(* CODESYS project PLS-logikk.project

Project tree, tasks and I/O mapping:
  Device : CODESYS Control Win V3 x64, CODESYS, version 3.5.21.50
    application Application
      libraries: Standard, 3.5.22.0 (System); Util, 3.5.22.0 (System); VisuDialogs, * (System); VisuElemBase, * (System); OpenWeather Client SL, * (CODESYS)
      task MainTask (cyclic, interval t#20ms, priority 1) calls PLC_PRG
      task VISU_TASK (cyclic, interval 100 ms, priority 31) calls VisuElems.Visu_Prg
      global variables GVL
      program PLC_PRG [ST]
      Lists/
        text list ValgtPIDVerdier
        text list Bakkesensor
        text list Energiventil
        text list Pumpe
      function block FB_Belimo_Energy_Valve [ST]
      function block safety_maks [ST]
      visualisation System_Overview
      visualisation System_Web_Configuration
      function block pumpe_ventil [ST]
      function block prognose [ST]
    EnergiVentilKommunikasjon : Ethernet, CODESYS, version 4.2.0.0
        settings: IPAddress = [192,168,0,1]; SubnetMask = [255,255,255,0]; GatewayAddress = [0,0,0,0]; MACAddress = [16#00,16#00,16#00,16#00,16#00,16#00]; SaveCommunicationSettings = FALSE; IPAddress = [192,168,0,2]; SubnetMask = [255,255,255,0]; GatewayAddress = [0,0,0,0]
      ModbusTCP_Server_Device : ModbusTCP Server Device, CODESYS, version 4.5.0.0
          settings: UpdateableHolding = TRUE
          unmapped channels: Holding Registers, Input Registers
      Modbus_TCP_Client : Modbus TCP Client, CODESYS, version 4.5.0.0
        Modbus_TCP_Server : Modbus TCP Server, CODESYS, version 4.5.0.0
            settings: Unit-ID = 255; IPAddress = [127, 0, 0, 1]; Channel 0.Function Code = 3; Channel 0.Read Offset = 16#0000; Channel 0.Read Length = 100; Channel 0.Write Offset = 0; Channel 0.Write Length = 0; Channel 0.Cycle Time = 100; Channel 1.Function Code = 16; Channel 1.Read Offset = 0; Channel 1.Read Length = 0; Channel 1.Write Offset = 16#0000; Channel 1.Write Length = 100; Channel 1.Cycle Time = 100
            input  Application.PLC_PRG.EnergiVentilRegs : ARRAY[0..99] OF WORD  // Channel 0
            output Application.GVL.DefaultEnergiVentilRegs : ARRAY[0..99] OF WORD  // Channel 1
    PumpeKommunikasjon : Ethernet, CODESYS, version 4.2.0.0
        settings: IPAddress = [192,168,0,1]; SubnetMask = [255,255,255,0]; GatewayAddress = [0,0,0,0]; MACAddress = [16#00,16#00,16#00,16#00,16#00,16#00]; SaveCommunicationSettings = FALSE; IPAddress = [192,168,0,2]; SubnetMask = [255,255,255,0]; GatewayAddress = [0,0,0,0]
      ModbusTCP_Server_Device_1 : ModbusTCP Server Device, CODESYS, version 4.5.0.0
          settings: Port = 503; UpdateableHolding = TRUE
          unmapped channels: Holding Registers, Input Registers
      Modbus_TCP_Client_1 : Modbus TCP Client, CODESYS, version 4.5.0.0
        Modbus_TCP_Server_1 : Modbus TCP Server, CODESYS, version 4.5.0.0
            settings: Unit-ID = 255; IPAddress = [127, 0, 0, 1]; Port = 503; Channel 0.Function Code = 3; Channel 0.Read Offset = 16#0000; Channel 0.Read Length = 100; Channel 0.Write Offset = 0; Channel 0.Write Length = 0; Channel 0.Cycle Time = 100; Channel 1.Function Code = 16; Channel 1.Read Offset = 0; Channel 1.Read Length = 0; Channel 1.Write Offset = 16#0000; Channel 1.Write Length = 100; Channel 1.Cycle Time = 100
            input  Application.PLC_PRG.PumpeRegs : ARRAY[0..99] OF WORD  // Channel 0
            output Application.GVL.DefaultPumpeRegs : ARRAY[0..99] OF WORD  // Channel 1
  libraries: VisuSymbols, 4.5.0.0 (System)
  text list GlobalTextList
  AC_GENERATOR_DATA
*)

// Device/Application/GVL
{attribute 'qualified_only'}
VAR_GLOBAL RETAIN
	
//system
energiventil_type : INT := 0; // 0 = Belimo, 1 = Siemens
bakkesensor_type  : INT := 0; //
pumpe_type        : INT := 0; //


//Simulering/falske variabler
DefaultEnergiVentilRegs: ARRAY[0..99] OF WORD;
DefaultPumpeRegs: ARRAY[0..99] OF WORD;
END_VAR

// Device/Application/PLC_PRG
PROGRAM PLC_PRG
VAR RETAIN
	

	EnergiVentilRegs: ARRAY[0..99] OF WORD;
	PumpeRegs: ARRAY[0..99] OF WORD;
	
	//prognose 
	fbWeather		: OPW.ForecastWeather;
	fbWeatherBatch	: OPW.ForecastWeatherBatch;

    xExecute		: BOOL;
    xError			: opw.ERROR;
	xDone			: BOOL;
	xbusy			: BOOL;
	location		: OPW.GeoLocation := (
		ws_city		:= "Tomsø",
		ws_country_code	:= "no",
		s_latitude	:= '69.6489',
		s_longitude	:= '18.9551'
	);
	eUnits			: OPW.UNIT_OPTION := OPW.UNIT_OPTION.METRIC;
	sLangugeCode	: OPW.LANGUAGE_CODE := 'en';
	
    apiKey			: STRING := '622d42f5e83be24b2235ae08787d5a43';

    idx				: INT;
		
	tFetch			: TON;
	
	prognose_temp				: ARRAY[0..23] OF REAL;
	prognose_nedbor				: ARRAY[0..23] OF REAL;
	prognose_vind				: ARRAY[0..23] OF REAL;
	
	// FBs
	Belimovalve : FB_Belimo_Energy_Valve;
	ventil0_regulering: safety_maks;
	smelte_regulering: pumpe_ventil;
	prognose_regulering: prognose;
	
	//styres av bruker
	veksler_temp_grense			: REAL:= 5;
	temp_beskyttelse_omraade	: REAL:= 5;
	min_temp_grense				: REAL:= -5;
	hysterese_C					: REAL:=1.5;
	smelte_grense				: REAL:=1.5;
	frost_grense				: REAL:=3;
	energi_grense				: REAL:=40;
	fukt_grense					: REAL:=40;
	
	Kp_array : ARRAY [0..2] OF REAL := [5,5,5]; // 0 = ventil0, 1 = pmp, 2 = ventiler
	Ti_array : ARRAY [0..2] OF REAL := [10,100,100];
	Td_array : ARRAY [0..2] OF REAL := [0,0,0];
	
	antall_soner				: INT:=3;
	bestemt_pumpe				: REAL:=50;
	min_pumpe					: REAL:=0;
	max_pumpe					: REAL:=100;
	bestemt_aapning				: ARRAY[1..20] OF REAL:= [20(0)];
	bestemt0_aapning			: REAL:= 0;
	
	ventil_min					: ARRAY[1..20] OF REAL:= [20(0)];
	ventil_maks					: ARRAY[1..20] OF REAL:= [20(100)];
	
	ventil0_min					: REAL:= 0;
	ventil0_maks				: REAL:= 100;
	
	manuell						: BOOL := FALSE;
	manuell0					: BOOL:= FALSE;
	reset						: ARRAY[1..20] OF BOOL:= [20(FALSE)];
	reset0						: BOOL:= FALSE;
	min_temp_aktiv				: BOOL:= TRUE;
	predikt						: BOOL:= FALSE;
	forvarme_horisont           : REAL:= 6.0;
	
	//interne variabler
	i							: INT := 0;
	pumpe_sone					: INT;
	varme_tap					: REAL;
	flow_sone					: REAL;
	tur_sone					: REAL;
	//Simulering (tall er kun eksempler)
	C1							: REAL:= 50000.0; // J/K
	C2							: REAL:= 80000.0; // J/K
	rho							: REAL:= 1000.0;  // kg/m^3
	c_1							: REAL:= 4186.0;  // J/(kg*K)
	
	Tx							: REAL:= 80;	  // C
	
	G1							: REAL:= 2000.0;  // W/K
	G2							: REAL:= 500.0;   // W/K
	G3							: REAL:= 300.0;   // W/K
	
	x5							: REAL:= 55;
	
	v1 							: REAL:= -5.0;
    v2 							: REAL:= 10.0;
    v3 							: REAL:= 10.0;
    v4 							: REAL:= 10.0;
	
	dx1							: REAL;
	dx2							: REAL;
	dx3							: REAL;
	dx4							: REAL;
	dx5							: REAL;
	deltat						: REAL:= 0.1;	  // s

	//output
	standby						: ARRAY[1..20] OF BOOL:= [20(FALSE)];
	running						: ARRAY[1..20] OF BOOL:= [20(FALSE)];
	lockout						: ARRAY[1..20] OF BOOL:= [20(FALSE)];
	tilstand                    : ARRAY[1..20] OF STRING;
	ventil0_aapning_cmd			: REAL;
	ventil_aapning_cmd			: ARRAY[1..20] OF REAL;
	pumpe_hastighet_cmd			: REAL;


	//innput
	tur_temp					: REAL;
	retur_temp					: REAL;
	retur_temp2					: REAL;
	ute_temp					: REAL := -10;
	energi_forbruk				: REAL;
	bakke_temp 					: ARRAY[1..20] OF REAL:= [20(5)];
    bakke_fukt 					: ARRAY[1..20] OF REAL:= [20(0)];
	ventil0_aapning_rd			: REAL;
	ventil_aapning_rd			: ARRAY[1..20] OF REAL;
	pumpe_hastighet_rd			: REAL;	
	
END_VAR


//init
CASE GVL.energiventil_type OF
0: Belimovalve(HoldingRegs := EnergiVentilRegs);
tur_temp := Belimovalve.temp1_C;
retur_temp := Belimovalve.temp2_C;
END_CASE

fbWeather(
    xExecute := xExecute,
	sApiKey := apiKey,
	pGeoLocation := ADR(location),
	eUnits := eUnits,
	data := fbWeatherBatch);
	
xError:= fbWeather.eError;
xDone:= fbWeather.xDone;
xbusy:= fbWeather.xBusy;

IF fbWeather.xDone THEN

    FOR i := 0 TO 23 DO

        prognose_temp[i] := fbWeatherBatch.aHourlyData[i].r_temperature;
        prognose_nedbor[i] := fbWeatherBatch.aHourlyData[i].r_snow_last_hour;
        prognose_vind[i] := fbWeatherBatch.aHourlyData[i].r_wind_speed;

    END_FOR
	
	xExecute := FALSE;

END_IF

tFetch(IN := TRUE, PT := T#60M);

IF tFetch.Q THEN
    xExecute := TRUE;
    tFetch(IN := FALSE);
END_IF

prognose_regulering(
    prognose_temp       := prognose_temp,
    prognose_nedbor     := prognose_nedbor,
    prognose_vind       := prognose_vind,
    ute_temp_na         := ute_temp,
    bakke_temp          := bakke_temp,

    base_frost_grense   := frost_grense,
	base_fukt_grense	:= fukt_grense,
    base_smelte_grense  := smelte_grense,
    base_min_pumpe      := min_pumpe,
    base_max_pumpe      := max_pumpe,

    forvarme_horisont   := forvarme_horisont,		// Se 6 timer frem
    maks_onsket_temp_okning := 3.0,		// Hev setpunkt med x antall grader
    grense_endring         := 2.0,		// Senk grensen med x antall grader
    min_pumpe_okning     := 15.0,	// Øk pumpe hastigheten for at hver sone alltid får nok strøm
	aktiver_prediktiv	:= predikt);



ventil0_regulering(
	retur_temp:= retur_temp,
	temp_grense:= veksler_temp_grense,
	temp_beskyttelse_omraade:= temp_beskyttelse_omraade,
	forbruk:= energi_forbruk,
	forbruk_grense:= energi_grense,
	bestemt_ventil:= bestemt0_aapning,
	Kp:= Kp_array[0],
	Ti:= Ti_array[0],
	Td:= Td_array[0],
	min_ventil:= ventil0_min,
	max_ventil:= ventil0_maks,
	manuell:= manuell0,
	reset:= reset0);

	
ventil0_aapning_cmd:= ventil0_regulering.ventil;


FOR i := 1 TO antall_soner DO
    IF smelte_regulering.running[i] THEN
        pumpe_sone := i;
    END_IF
END_FOR
i:=0;

smelte_regulering(
	antall_soner:= antall_soner,
	bakke_temp:=bakke_temp,
	bakke_fukt:= bakke_fukt,
	frost_grense:= frost_grense,
	smelte_grense:= smelte_grense,
	fukt_grense:= fukt_grense,
	hysterese:= hysterese_C,
	min_temp_grense:= min_temp_grense,
	min_temp_aktiv:= min_temp_aktiv,
	Kp_pmp:= Kp_array[1],
	Tn_pmp:= Ti_array[1],
	Tv_pmp:= Td_array[1],
	Kp_vnt:= Kp_array[2],
	Tn_vnt:= Ti_array[2],
	Tv_vnt:= Td_array[2],
	manuell:= manuell,
	reset:= reset,
	bestemt_pumpe:= bestemt_pumpe,
	min_pumpe:= min_pumpe,
	max_pumpe:= max_pumpe,
	pumpe_sone:= pumpe_sone,
	bestemt_aapning:=bestemt_aapning,
	ventil_min:= ventil_min,
	ventil_maks:= ventil_maks);

standby:= smelte_regulering.standby;
running:= smelte_regulering.running;
lockout:= smelte_regulering.min_temp_lockout;
ventil_aapning_cmd:= smelte_regulering.ventil_cmd;
pumpe_hastighet_cmd:= smelte_regulering.pumpe_cmd;


FOR i := 1 TO antall_soner DO
	IF standby[i] THEN 
		tilstand[i] := 'i standby';
	ELSIF running[i] THEN 
		tilstand[i] := 'i running';
	ELSIF lockout[i] THEN 
		tilstand[i] := 'i lockout';
	ELSE
		tilstand[i] := 'av';
	END_IF
END_FOR

//simulering
	retur_temp:= ((1.0/ventil0_aapning_rd - 1.0) * tur_temp 
	+ ventil_aapning_rd[1] * v2 + ventil_aapning_rd[2] * ventil_aapning_rd[2] * v3 
	+ (1.0 - ventil_aapning_rd[1] - ventil_aapning_rd[1] * ventil_aapning_rd[2]) * v4);
	
	
dx1 := (1.0/C1) * ( pumpe_hastighet_rd * rho * c_1 * ( Tx - tur_temp) - G1 * (tur_temp - x5));

dx2 := (1.0/C2) * ( pumpe_hastighet_rd * ventil0_aapning_rd * ventil_aapning_rd[1] * rho * c_1 * (tur_temp - v2) + G2 * (v2 - bakke_temp[1]) - G3 * (bakke_temp[1] - ute_temp));

dx3 := (1.0/C2) * ( pumpe_hastighet_rd * ventil0_aapning_rd * ventil_aapning_rd[1] * ventil_aapning_rd[2] * rho * c_1 * (tur_temp - v3) + G2 * (v3 - bakke_temp[2]) - G3 * (bakke_temp[2] - ute_temp));

dx4 := (1.0/C2) * ( pumpe_hastighet_rd * ventil0_aapning_rd * (1.0 - ventil_aapning_rd[1] - ventil_aapning_rd[1]*ventil_aapning_rd[2]) * rho * c_1 * (tur_temp - v4) + G2 * (v4 - bakke_temp[3]) - G3 * (bakke_temp[3] - ute_temp));

dx5 := (1.0/C1) * ( pumpe_hastighet_rd * rho * c_1 * (retur_temp- x5) - G1 * (x5 - tur_temp));

//Numerisk integrasjon (Euler)
tur_temp := tur_temp + dx1 * deltat;
bakke_temp[1] := bakke_temp[1] + dx2 * deltat;
bakke_temp[2] := bakke_temp[2] + dx3 * deltat;
bakke_temp[3] := bakke_temp[3] + dx4 * deltat;
x5 := x5 + dx5 * deltat;

//Enkel beregning av temperaturen ut av hver sone
v2 := tur_temp - (tur_temp - bakke_temp[1]* pumpe_hastighet_rd * ventil0_aapning_rd * ventil_aapning_rd[1]);
v3 := tur_temp - (tur_temp - bakke_temp[1]* pumpe_hastighet_rd * ventil0_aapning_rd * ventil_aapning_rd[1] * ventil_aapning_rd[2]);
v4 := tur_temp - (tur_temp - bakke_temp[1]* pumpe_hastighet_rd * ventil0_aapning_rd * (1.0 - ventil_aapning_rd[1] - ventil_aapning_rd[1]*ventil_aapning_rd[2]));

END_PROGRAM

// Device/Application/prognose
FUNCTION_BLOCK prognose
VAR_INPUT
    // ── Værvarselsdata fra Python (oppdateres f.eks. hvert 30. minutt) ──────
    // Timevis prognose, indeks 0 = neste hele time, 23 = 24 timer frem
    prognose_temp       : ARRAY[0..23] OF REAL;		// Utetemperatur [°C]
    prognose_nedbor     : ARRAY[0..23] OF REAL;		// Nedbørsmengde [mm/t]
    prognose_vind       : ARRAY[0..23] OF REAL;		// Vindhastighet [m/s]

    // ── Nåtilstand ──────────────────────────────────────────────────────────
    ute_temp_na         : REAL;                     // Faktisk utetemperatur nå [°C]
    bakke_temp          : ARRAY[1..20] OF REAL;     // Faktisk bakketemperatur per sone [°C]

    // ── Brukerens grunninnstillinger (pass-through når prediktiv er av) ─────
    base_frost_grense   : REAL;     // Normal frostgrense for å gå i standby [°C]
    base_smelte_grense  : REAL;     // Normal smeltegrense for å gå i running [°C]
	base_fukt_grense	: REAL;		// Normal fuktgrense for å gå i running [%]
    base_min_pumpe      : REAL;     // Normalt minimum pumpesignal [%]
    base_max_pumpe      : REAL;     // Normalt maksimum pumpesignal [%]

    // ── Prediktive tuningsparametre ──────────────────────────────────────────
    forvarme_horisont   : REAL := 6.0;	// Hvor mange timer frem vi ser etter snøhendelser [t] Anbefalt: 3–8 t avhengig av termisk tregheten til banen
    maks_onsket_temp_okning : REAL := 3.0;	// Hvor mye vi hever onsket_temp under forvarmning [°C] Heves gradvis jo nærmere snøhendelsen er
    grense_endring         : REAL := 1.5;	// Hvor mye vi hever frost_grense / smelte_grense for tidlig aktivering [°C] Gjør at sonene starter standby/running litt tidligere enn normalt
    min_pumpe_okning     : REAL := 15.0;	// Ekstra minimum pumpeprosent under forvarmning [%] Hindrer at pumpen stopper helt mens banen forvarmes
    vind_kjoele_faktor  : REAL := 0.16;	// Justeringsfaktor for vindavkjøling (standard vindkjøleformel) Følger wind chill index
    aktiver_prediktiv   : BOOL := FALSE;	// Slå prediktiv styring av/på
END_VAR

VAR_OUTPUT
    // ── Justerte setpunkter – kobles direkte til smelte_regulering ──────────
    ut_frost_grense     : REAL;     // Justert frostgrense
    ut_smelte_grense    : REAL;     // Justert smeltegrense
	ut_fukt_grense		: REAL;		// Justert fuktgrense
    ut_min_pumpe        : REAL;     // Justert minimum pumpe
    ut_max_pumpe        : REAL;     // Uendret, sendt videre

    // ── Statusinformasjon ────────────────────────────────────────────────────
    snoe_risiko         : REAL;     // Beregnet snørisiko 0–100
    timer_til_sno		: REAL;     	// Timer til første forventede snøhendelse (-1 = ingen)
    forvarme_aktiv		: BOOL;     // TRUE mens prediktiv forvarmning pågår
    forvarme_intensitet : REAL;     // 0–100 % — hvor aggressivt vi forvarmer
    vind_prognose_temp	: ARRAY[0..23] OF REAL;     	// Beregnet vindkjølt temperatur [°C]
END_VAR

VAR
    i                   : INT;

    // Interne beregningsvariabler
    forste_sno_time    : REAL;     // Indeks (timer) til første snøhendelse
    sno_funnet         : BOOL;
    sum_sno_mm         : REAL;     // Total forventet snønedbør innen horisonten
    min_prognose_temp   : REAL;     // Laveste temperatur innen horisonten

    intensitet_raa      : REAL;     // Ubehandlet intensitetsverdi 0–1
    tid_igjen_normert   : REAL;     // 0 = snøen er her, 1 = akkurat innenfor horisont
    temp_bidrag         : REAL;
    nedbor_bidrag       : REAL;
    vind_bidrag         : REAL;
    horisont_heltall    : INT;      // Horisont avrundet til heltall timer (maks 23)
END_VAR

//Beskytte mot dårlig input
IF forvarme_horisont < 1.0 THEN forvarme_horisont := 1.0; END_IF
IF forvarme_horisont > 23.0 THEN forvarme_horisont := 23.0; END_IF
horisont_heltall := REAL_TO_INT(forvarme_horisont);

//Finner første snøhendelse, total snø, laveste temp
sno_funnet      := FALSE;
forste_sno_time := -1.0;
sum_sno_mm      := 0.0;
min_prognose_temp := prognose_temp[0];

FOR i := 0 TO horisont_heltall DO
	//Regner ut hvor mye vinden påvirker temperaturen
	IF prognose_vind[i] > 1.3 AND prognose_temp[i] < 10.0 THEN
    	vind_prognose_temp[i] := 13.12
					 			+ 0.6215  * prognose_temp[i]
								- 11.37   * EXPT(prognose_vind[i] * 3.6, vind_kjoele_faktor)
								+ 0.3965  * prognose_temp[i] * EXPT(prognose_vind[i] * 3.6, vind_kjoele_faktor);
	ELSE
		vind_prognose_temp[i] := prognose_temp[i];
	END_IF

    // Registrer laveste temperatur 
    IF vind_prognose_temp[i] < min_prognose_temp THEN
        min_prognose_temp := vind_prognose_temp[i];
    END_IF

    // Finner ut om det kommer snø basert på forventet nedbør og temperatur
    IF (vind_prognose_temp[i] <= 0 AND prognose_nedbor[i] > 0.1) THEN

        sum_sno_mm := sum_sno_mm + prognose_nedbor[i];

        IF NOT sno_funnet THEN
            forste_sno_time := INT_TO_REAL(i);
            sno_funnet := TRUE;
        END_IF
	END_IF
END_FOR

timer_til_sno := forste_sno_time;  // -1 hvis ingen hendelse funnet

// Risiko bergening  (0–100)%
//    Tre bidrag vektet sammen:
//      – Temperaturrisiko : lavere temp → høyere risiko
//      – Nedbørsrisiko    : mer nedbør → høyere risiko
//      – Vindrisiko       : sterk vind forsterker nedkjøling

// Temperaturbidrag: 0 ved +5 °C eller mer, 100 ved -10 °C eller mindre
temp_bidrag := LIMIT(0.0, (5.0 - min_prognose_temp) / 15.0 * 100.0, 100.0);

// Nedbørsbidrag: 0 ved 0 mm eller mindre, 100 ved ≥10 mm total nedbør i vinduet
nedbor_bidrag := LIMIT(0.0, sum_sno_mm / 10.0 * 100.0, 100.0);

// Vindbidrag: 0 ved 0 m/s eller mindre, 100 ved ≥15 m/s
vind_bidrag := LIMIT(0.0, prognose_vind[0] / 15.0 * 100.0, 100.0);

// Vektet sum  (temperatur teller mest for bakke-systemet)
snoe_risiko := LIMIT(0.0,
    0.50 * temp_bidrag
  + 0.35 * nedbor_bidrag
  + 0.15 * vind_bidrag,
  100.0);

// Beregner forvarme intensitet  (0–1 brukes videre, 0–100 for å vise bruker)
//    Intensiteten trappes opp jo nærmere snøhendelsen vi er.
//    Ingen snøhendelse innen horisonten gjør at intensitet = 0
intensitet_raa := 0.0;

IF aktiver_prediktiv AND sno_funnet THEN
    // Normaliser: 0 = snøen er her, 1 = akkurat på horisonten
    tid_igjen_normert := LIMIT(0.0, forste_sno_time / forvarme_horisont, 1.0);

    // Lineær opptrapping: tidligst = 30 % intensitet, nærmer seg = 100 %
    intensitet_raa := LIMIT(0.0, 1.0 - (0.7 * tid_igjen_normert), 1.0);

    // I tillegg skaleres med risikoscoren (sterk storm → enda mer aggressiv)
    intensitet_raa := intensitet_raa * (0.5 + 0.5 * (snoe_risiko / 100.0));
END_IF

forvarme_aktiv      := intensitet_raa > 0.0;
forvarme_intensitet := LIMIT(0.0, intensitet_raa * 100.0, 100.0);

// Justerer sett punkter
//    Alle utganger faller tilbake til brukerens basisverdier når prediktiv er av
//    eller ingen snø er forventet.
IF aktiver_prediktiv AND forvarme_aktiv THEN

    // Hev frost-, fukt- og smeltegrensene litt slik at sonene aktiverer seg tidligere
    ut_frost_grense  := base_frost_grense  + grense_endring * intensitet_raa;
    ut_smelte_grense := base_smelte_grense + grense_endring * intensitet_raa;
	ut_fukt_grense   := base_fukt_grense   - base_fukt_grense * intensitet_raa;

    // Hev minimum pumpe for å hindre pumpen i å stoppe under forvarmning
    ut_min_pumpe     := LIMIT(base_min_pumpe,
                              base_min_pumpe + min_pumpe_okning * forvarme_intensitet,
                              base_max_pumpe * 0.8);
    ut_max_pumpe     := base_max_pumpe;

ELSE
    // Pass-through når prediktiv styring gjør ingenting (enten ved avskrudd eller ved ingen forventet snø)
    ut_frost_grense  := base_frost_grense;
    ut_smelte_grense := base_smelte_grense;
	ut_fukt_grense	 := base_fukt_grense;
    ut_min_pumpe     := base_min_pumpe;
    ut_max_pumpe     := base_max_pumpe;
END_IF

END_FUNCTION_BLOCK

// Device/Application/FB_Belimo_Energy_Valve
FUNCTION_BLOCK FB_Belimo_Energy_Valve
VAR_INPUT
	HoldingRegs : ARRAY[0..99] OF WORD; // map til Modbus Holding Registers
END_VAR
VAR_OUTPUT
	RelPos_pct : REAL;
    Flow_lps : REAL;
    Temp1_C : REAL;
    Temp2_C : REAL;
    DeltaT_K : REAL;
    Energy_kWh : REAL;
END_VAR
VAR
	rawLow : WORD;
    rawHigh : WORD;
    raw32 : DWORD;
END_VAR


//Konvertering
RelPos_pct := TO_REAL(HoldingRegs[4]) * 0.01;

Flow_lps := TO_REAL(HoldingRegs[7]) * 0.001;

Temp1_C := TO_REAL(HoldingRegs[19]) * 0.01; //vi sier at dette er tur temp for enkelhet, kunne ha vært invertert

Temp2_C := TO_REAL(HoldingRegs[21]) * 0.01;// retur temp

DeltaT_K := TO_REAL(HoldingRegs[23]) * 0.01;// diff mellom tur og retur

END_FUNCTION_BLOCK

// Device/Application/safety_maks
FUNCTION_BLOCK safety_maks
VAR_INPUT
	retur_temp                  : REAL;  // Retur temperatur sensor rett før varmeveksler og etter treveis ventil
    temp_grense                 : REAL;  // Temperatur hvor man må begynne å ta hensyn til sikkerheten rundt varmevekslere
    temp_beskyttelse_omraade    : REAL;  // Området under tem_grense for helt stengt ventil
                                         // Ved temp_grense - temp_beskyttelse_omraade blir ventil = 100%

    forbruk                     : REAL;  // Nåverende energi forbruk (kW)
    forbruk_grense              : REAL;  // Maks tillat energi forbruk (kW)

    bestemt_ventil              : REAL;  // Hvor stor åpning ventilen har i manuell modus
    Kp                          : REAL;  
    Ti                          : REAL;
    Td                          : REAL;
    min_ventil                  : REAL; // Når ventilen går fullt til smelte soner
    max_ventil                  : REAL; // Når ventilen går fullt tilbake til varmeveklser
    manuell                     : BOOL;
    reset                       : BOOL;
END_VAR
VAR_OUTPUT
    ventil                      : REAL;	// Signal som bestemmer ventil possisjon
    beskyttelse_aktiv           : BOOL; // På når beskyttelse modus er aktiv
    beskyttelse_faktor          : REAL; // Faktor som sier hvor mye beskytelsen er på (0.0 beskyttelsen er av, 1.0 beskyttelsen sender alt tilbake til varmeveksler
END_VAR
VAR
	offset                      : REAL := 0;
    pid                         : PID;
    Max_tillatt                : REAL;  // Min valve position allowed by protection
END_VAR

// BESKYTT MOT DÅRLIG INNGANG
// Forhindrer divisjon med null hvis område ikke er konfigurert
IF temp_beskyttelse_omraade <= 0.0 THEN
    temp_beskyttelse_omraade := 1.0;
END_IF

//bestemmer hvor mye beskyttelse som skla være på
IF retur_temp >= temp_grense THEN
    beskyttelse_faktor := 0.0;
ELSIF retur_temp <= (temp_grense - temp_beskyttelse_omraade) THEN
    beskyttelse_faktor := 1.0;
ELSE
    beskyttelse_faktor := (temp_grense - retur_temp) / temp_beskyttelse_omraade;
END_IF;

//setter beskytelses indikator på hvis det er mer enn 0.0 beskytelse
beskyttelse_aktiv := beskyttelse_faktor > 0.0;

//definerer en minimums grense tillat slik at pid-regulatoren ikke kan sende mer til smelte soner enn trygt
Max_tillatt := max_ventil - (beskyttelse_faktor * (max_ventil - min_ventil));

//pid for å regulere energi forbruk
pid(
    ACTUAL      := forbruk,
    SET_POINT   := forbruk_grense,
    KP          := Kp,
    TN          := Ti,
    TV          := Td,
    Y_MANUAL    := bestemt_ventil,
    Y_OFFSET    := offset,
    Y_MIN       := min_ventil,
    Y_MAX       := max_tillatt,
    MANUAL      := manuell,
    RESET       := reset);

ventil := LIMIT(Min_ventil, pid.Y, max_tillatt);

//når ventil er 100% går all strøm til smelte sonene og når ventil er 0% vil alø strøm gå igjennom tre veis ventilen og tilbake til varmeveksleren

END_FUNCTION_BLOCK

// Device/Application/pumpe_ventil
FUNCTION_BLOCK pumpe_ventil
VAR_INPUT
	
	antall_soner        : INT;	//Hvor mange soner du ønsker å regulere
    bakke_temp          : ARRAY[1..20] OF REAL;	//Array av alle bakke temp målinger
    bakke_fukt          : ARRAY[1..20] OF REAL;	//Array av alle bakke fukt målinger
	
    frost_grense        : REAL;	//Nedre grense for å starte tining
    smelte_grense       : REAL;	//Øvre grense for å starte tining
    fukt_grense         : REAL;	//Grense for hvor mye fukt for å starte tining
    hysterese           : REAL;	//Ekstra ledd for å forhindre hopping mellom tilstander
	
	min_temp_grense     : REAL;	//Under denne tempen vil systemet gå i lockout
    min_temp_aktiv      : BOOL; //Velg om du vil inkludere lockout
	
	Kp_pmp              : REAL;	//Kp-verdi for pumpe
    Tn_pmp              : REAL;	//Tn-verdi for pumpe
    Tv_pmp              : REAL;	//Tv-verdi for pumpe
	Kp_vnt              : REAL;	//Kp-verdi for ventil
    Tn_vnt              : REAL;	//Tn-verdi for ventil
    Tv_vnt              : REAL;	//Tv-verdi for ventil
    manuell             : BOOL;	//Array av valg der bruker bestemer om sonen skal være i manuell modus
    reset               : ARRAY[1..20] OF BOOL;	//Reset for integral delen av regulatorer for hver sone

	bestemt_pumpe       : REAL;	//Verdi pumpen går til når den er i manuell modus
    min_pumpe           : REAL;	//Minimum pumpe verdi
    max_pumpe           : REAL;	//Maximimum pumpe verdi
    pumpe_sone          : INT;	//Sone som skal reguleres av pumpen

	bestemt_aapning     : ARRAY[1..20] OF REAL;	//Verdi ventilen i hver sone går til når den er i manuell modus
	ventil_min          : ARRAY[1..20] OF REAL;	//Minimum ventil verdi
	ventil_maks         : ARRAY[1..20] OF REAL;	//Maximum ventil verdi

END_VAR
VAR_OUTPUT
	standby             : ARRAY[1..20] OF BOOL;	//På når sonen er i standby modus
	running             : ARRAY[1..20] OF BOOL;	//På når sonen er i running modus
	ventil_cmd          : ARRAY[1..20] OF REAL;	//Signal som bestemmer ventil sin åpning
	pumpe_cmd           : REAL;	//Signal som bestemmer pumpe sin hastighet i prosent
	min_temp_lockout    : ARRAY[1..20] OF BOOL; //På når sonen er i lockout modus

END_VAR
VAR
	i					: INT;
    sone_case			: ARRAY[1..20] OF INT:= [20(0)]; // 0=AV 1=STANDBY 2=RUNNING 3=LOCKOUT
    pid_ventil          : ARRAY[1..20] OF PID;
    pid_pumpe           : PID;
    Lockout            	: ARRAY[1..20] OF BOOL;
	offset_pmp          : REAL := 0;	//Offset-verdi for pumpe
    offset_vnt          : REAL := 0; //Offset-verdi for ventil
END_VAR

FOR i := 1 TO antall_soner DO


 Lockout[i] := min_temp_aktiv AND (bakke_temp[i] < min_temp_grense) AND NOT manuell;
 
	IF Lockout[i] THEN 
        sone_case[i] := 3;
    ELSIF sone_case[i] = 3 THEN
        // Gå kun ut av lockout hvis temp er over min temp grense + en hysterese
        IF NOT min_temp_aktiv OR bakke_temp[i] >= (min_temp_grense + hysterese) THEN
            sone_case[i] := 0; // send tilbake til state maskinen for videre valg
        END_IF
    END_IF;

    // Kjører kun hvis sonen ikke er i lockout
   	IF sone_case[i] <> 3 THEN

        CASE sone_case[i] OF

            0: // AV
                IF bakke_temp[i] <= frost_grense THEN
                    sone_case[i] := 1;
                END_IF

            1: // STANDBY
                IF bakke_fukt[i] > fukt_grense AND bakke_temp[i] <= smelte_grense THEN
					reset[i] := TRUE;
					reset[i] := FALSE;
                    sone_case[i] := 2;
                ELSIF bakke_temp[i] > (frost_grense + hysterese) THEN
					reset[i] := TRUE;
					reset[i] := FALSE;
                    sone_case[i] := 0;
                END_IF

            2: // RUNNING
			
                IF bakke_fukt[i] <= (fukt_grense + hysterese) OR bakke_temp[i] > (smelte_grense + hysterese)THEN
					reset[i] := TRUE;
					reset[i] := FALSE;
                    sone_case[i] := 1;
                END_IF

        END_CASE;
	
	END_IF;

    // Gir bruker info om hvilken modus sonen er i
    standby[i]          := (sone_case[i] = 1);
    running[i]          := (sone_case[i] = 2);
    min_temp_lockout[i] := (sone_case[i] = 3);

	
	//Bestemmer ventil og pumpe signal basert på hvilken modus sonen er i
    CASE sone_case[i] OF

        0: // OFF
            ventil_cmd[i] := 0;
			//fjern denne PIDen?
            pid_ventil[i](
                ACTUAL      := bakke_temp[i],
                SET_POINT   := 0,
                KP:= Kp_vnt, TN:= Tn_vnt, TV:= Tv_vnt,
                Y_MANUAL    := 0,
                Y_OFFSET    := 0,
                Y_MIN       := ventil_min[i],
                Y_MAX       := ventil_maks[i],
                MANUAL      := TRUE,
                RESET       := TRUE);

        1: // STANDBY
            pid_ventil[i](
                ACTUAL      := bakke_temp[i],
                SET_POINT   := (frost_grense + hysterese),
                KP:= Kp_vnt, TN:= Tn_vnt, TV:= Tv_vnt,
                Y_MANUAL    := bestemt_aapning[i],
                Y_OFFSET    := offset_vnt,
                Y_MIN       := ventil_min[i],
                Y_MAX       := ventil_maks[i],
                MANUAL      := manuell,
                RESET       := reset[i]);
            ventil_cmd[i] := pid_ventil[i].Y;

        2: // RUNNING
            IF i = pumpe_sone THEN
                ventil_cmd[i] := ventil_maks[i];
                pid_pumpe(
                    ACTUAL      := bakke_temp[i],
                    SET_POINT   := (smelte_grense + hysterese),
                    KP:= Kp_pmp, TN:= Tn_pmp, TV:= Tv_pmp,
                    Y_MANUAL    := bestemt_pumpe,
                    Y_OFFSET    := offset_pmp,
                    Y_MIN       := min_pumpe,
                    Y_MAX       := max_pumpe,
                    MANUAL      := manuell,
                    RESET       := reset[i]);
                pumpe_cmd := pid_pumpe.Y;
            ELSE
                pid_ventil[i](
                    ACTUAL      := bakke_temp[i],
                    SET_POINT   := (smelte_grense + hysterese),
                    KP:= Kp_vnt, TN:= Tn_vnt, TV:= Tv_vnt,
                    Y_MANUAL    := bestemt_aapning[i],
                    Y_OFFSET    := offset_vnt,
                    Y_MIN       := ventil_min[i],
                    Y_MAX       := ventil_maks[i],
                    MANUAL      := manuell,
                    RESET       := reset[i]);
                ventil_cmd[i] := pid_ventil[i].Y;
            END_IF

        3: // LOCKOUT - Fungerer som av, reset alt
            ventil_cmd[i] := 0;
			//fjern PIDen?
            pid_ventil[i](
                ACTUAL      := bakke_temp[i],
                SET_POINT   := 0,
                KP:= Kp_vnt, TN:= Tn_vnt, TV:= Tv_vnt,
                Y_MANUAL    := 0,
                Y_OFFSET    := 0,
                Y_MIN       := ventil_min[i],
                Y_MAX       := ventil_maks[i],
                MANUAL      := TRUE,
                RESET       := TRUE);

    END_CASE;

END_FOR;
i:=1;

// Bestemmer Pumpe signal når pumpe sone er i standby og når det ikke er noen pumpe sone
IF pumpe_sone < 1 OR pumpe_sone > antall_soner THEN
    pumpe_cmd := 0;
ELSIF sone_case[pumpe_sone] = 0 THEN
    pumpe_cmd := 0;
ELSIF sone_case[pumpe_sone] = 1 OR sone_case[pumpe_sone] = 3 THEN //Vil dette funke? Setter pumpen til minimum når pumpe sonen enten er i lockout eller standby
    pumpe_cmd := min_pumpe;
END_IF;

END_FUNCTION_BLOCK

// Device/Application/System_Overview
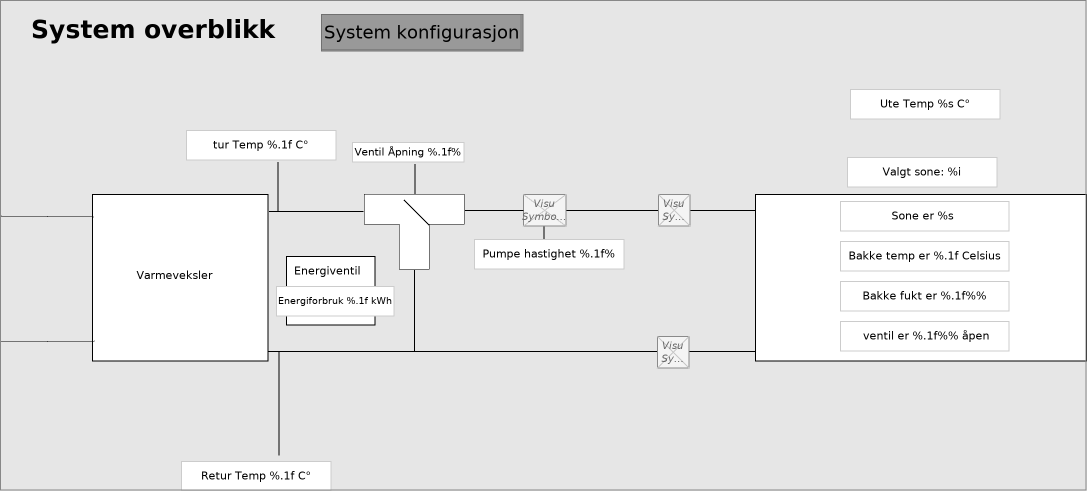
VISUALIZATION System_Overview  // 1087x491
VAR
valgt_sone: INT:=1;	
END_VAR
    Line (544,246) (544,216)
    Line (268,351) (762,351)
    Line (566,210) (761,210)
    RoundedRectangle (755,194 332x167)
    Rectangle (92,194 176x167)
    Label (99,256 151x39), "Varmeveksler"
    Line (93,217) (1,216)
    Line (94,341) (0,342)
    Polygon (364,194) (464,194) (464,224) (429,224) (429,269) (399,269) (399,224) (364,224)
    Line (429,225) (404,200)
    Textfield (352,142 112x20), "Ventil Åpning %.1f%", tooltip "0% = tur går direkte til retur, 100% = tur går videre til smeltesoner", text variable: PLC_PRG.ventil0_aapning_cmd
    Image (523,194 43x32), image: VisuSymbols.Symbols.ArrowBoldRight
    Textfield (474,239 150x30), "Pumpe hastighet %.1f%", text variable: PLC_PRG.pumpe_hastighet_cmd
    Line (269,211) (363,211)
    Rectangle (286,256 89x69)
    Label (280,256 95x30), "Energiventil"
    Textfield (276,286 118x30), "Energiforbruk %.1f kWh", text variable: PLC_PRG.energi_forbruk
    Line (414,270) (414,351)
    Line (465,210) (523,210)
    Line (279,455) (279,352)
    Textfield (181,461 150x30), "Retur Temp %.1f C°", text variable: PLC_PRG.retur_temp
    Line (415,194) (415,164)
    Textfield (186,130 150x30), "tur Temp %.1f C°", text variable: PLC_PRG.tur_temp
    Line (278,211) (278,162)
    Textfield (847,157 150x30), "Valgt sone: %i", text variable: valgt_sone
        OnMouseClick: write the text variable via VisuDialogs.Numpad, min 1, max PLC_PRG.antall_soner
    Textfield (840,241 169x30), "Bakke temp er %.1f Celsius", text variable: PLC_PRG.bakke_temp[valgt_sone]
    Textfield (840,281 169x30), "Bakke fukt er %.1f%%", text variable: PLC_PRG.bakke_fukt[valgt_sone]
    Button (321,14 202x37), "System konfigurasjon"
        OnMouseClick:  Assign=System_Web_Configuration, Type=Assignment
    Label (5,14 296x30), "System overblikk"
    Image (657,336 32x32), image: VisuSymbols.Symbols.ArrowBack
    Image (658,194 32x32), angle 180, image: VisuSymbols.Symbols.ArrowBack
    Textfield (840,321 169x30), "ventil er %.1f%% åpen", text variable: PLC_PRG.ventil_aapning_cmd[valgt_sone]
    Textfield (850,89 150x30), "Ute Temp %s C°", text variable: PLC_PRG.ute_temp
    Textfield (840,201 169x30), "Sone er %s", text variable: PLC_PRG.tilstand[valgt_sone]
END_VISUALIZATION

// Device/Application/System_Web_Configuration
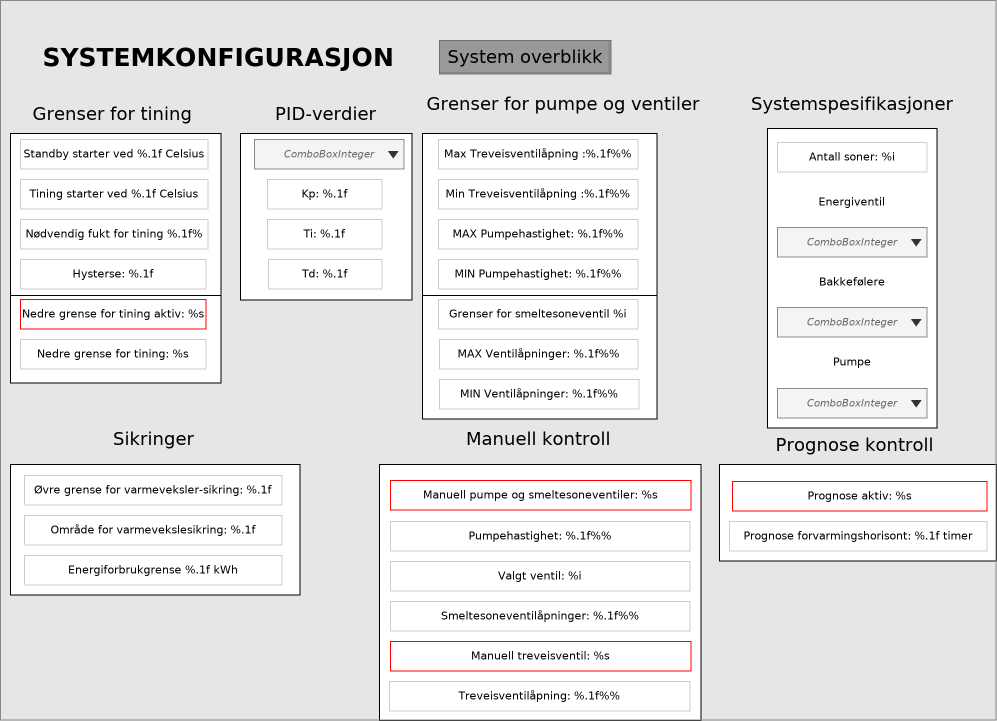
VISUALIZATION System_Web_Configuration  // 997x721
VAR
valgt_pid : INT := 0;
valgt_ventil: INT :=1;
END_VAR
    RoundedRectangle (719,464 278x97)
    RoundedRectangle (379,464 322x257)
    RoundedRectangle (767,128 170x300)
    RoundedRectangle (10,464 290x131)
    RoundedRectangle (422,133 235x286)
    RoundedRectangle (422,295 235x124)
    RoundedRectangle (10,133 211x250)
    RoundedRectangle (10,295 211x88)
    RoundedRectangle (240,133 172x167)
    Textfield (20,179 188x30), "Tining starter ved %.1f Celsius", text variable: PLC_PRG.smelte_grense
        OnMouseClick: write the text variable via VisuDialogs.Numpad
    Label (34,99 157x30), "Grenser for tining"
    Textfield (20,139 188x30), "Standby starter ved %.1f Celsius", text variable: PLC_PRG.frost_grense
        OnMouseClick: write the text variable via VisuDialogs.Numpad
    Textfield (267,179 115x30), "Kp: %.1f", text variable: PLC_PRG.Kp_array[valgt_pid]
        OnMouseClick: write the text variable via VisuDialogs.Numpad
    Textfield (267,219 115x30), "Ti: %.1f", text variable: PLC_PRG.Ti_array[valgt_pid]
        OnMouseClick: write the text variable via VisuDialogs.Numpad
    Label (247,99 157x30), "PID-verdier"
    Textfield (268,259 114x30), "Td: %.1f", text variable: PLC_PRG.Td_array[valgt_pid]
        OnMouseClick: write the text variable via VisuDialogs.Numpad
    Textfield (24,555 258x30), "Energiforbrukgrense %.1f kWh", tooltip "Treveisventilen vil bli regulert etter denne grensen, varmeveksler-sikring har en høyere prioritet", text variable: PLC_PRG.energi_grense
        OnMouseClick: write the text variable via VisuDialogs.Numpad
    Textfield (20,219 188x30), "Nødvendig fukt for tining %.1f%", text variable: PLC_PRG.fukt_grense
        OnMouseClick: write the text variable via VisuDialogs.Numpad
    Textfield (390,480 301x30), "Manuell pumpe og smeltesoneventiler: %s", tooltip "skru manuell styring av/på", text variable: PLC_PRG.manuell
        toggle PLC_PRG.manuell
    Label (421,424 235x30), "Manuell kontroll"
    Textfield (390,521 300x30), "Pumpehastighet: %.1f%%", text variable: PLC_PRG.bestemt_pumpe
        OnMouseClick: write the text variable via VisuDialogs.Numpad, min 0, max 100
    Textfield (390,601 300x30), "Smeltesoneventilåpninger: %.1f%%", text variable: PLC_PRG.bestemt_aapning[valgt_ventil]
        OnMouseClick: write the text variable via VisuDialogs.Numpad, min 0, max 100
    Textfield (777,142 150x30), "Antall soner: %i", text variable: PLC_PRG.antall_soner
        OnMouseClick: write the text variable via VisuDialogs.Numpad, min 1, max 20
    Line (0,154)
    Textfield (438,259 200x30), "MIN Pumpehastighet: %.1f%%", text variable: PLC_PRG.min_pumpe
        OnMouseClick: write the text variable via VisuDialogs.Numpad, min 0, max PLC_PRG.max_pumpe
    Textfield (438,219 200x30), "MAX Pumpehastighet: %.1f%%", text variable: PLC_PRG.max_pumpe
        OnMouseClick: write the text variable via VisuDialogs.Numpad, min PLC_PRG.min_pumpe, max 100
    Textfield (439,379 200x30), "MIN Ventilåpninger: %.1f%%", tooltip "Ventilåpning for standby og minimumsgrense for tining", text variable: PLC_PRG.ventil_min[valgt_ventil]
        OnMouseClick: write the text variable via VisuDialogs.Numpad, min 0, max PLC_PRG.ventil_maks[valgt_ventil]
    Textfield (439,339 199x30), "MAX Ventilåpninger: %.1f%%", tooltip "Ventilåpning for standby og maximumsgrense for tining", text variable: PLC_PRG.ventil_maks[valgt_ventil]
        OnMouseClick: write the text variable via VisuDialogs.Numpad, min PLC_PRG.ventil_min[valgt_ventil], max 100
    ComboBoxInteger (777,227 150x30), tooltip "Funksjonelt ubrukt for nå, ideen er å vise hvor enkelt det ville ha vært å velge ventil, sensor og pumpe", variable: GVL.energiventil_type, text list: 'Energiventil'
    ComboBoxInteger (777,307 150x30), tooltip "Funksjonelt ubrukt for nå, ideen er å vise hvor enkelt det ville ha vært å velge ventil, sensor og pumpe", variable: GVL.bakkesensor_type, text list: 'Bakkesensor'
    Label (5,5 427x104), "SYSTEMKONFIGURASJON"
    Label (425,89 276x30), "Grenser for pumpe og ventiler"
    Label (737,89 230x30), "Systemspesifikasjoner"
    Label (777,187 150x30), "Energiventil"
    Label (777,267 150x30), "Bakkefølere"
    Label (777,347 150x30), "Pumpe"
    ComboBoxInteger (777,388 150x30), tooltip "Funksjonelt ubrukt for nå, ideen er å vise hvor enkelt det ville ha vært å velge ventil, sensor og pumpe", variable: GVL.pumpe_type, text list: 'Pumpe'
    Button (439,40 172x34), "System overblikk"
        OnMouseClick:  Assign=System_Overview, Type=Assignment
    Textfield (20,259 186x30), "Hysterse: %.1f", tooltip "Hysteresen gjelder når reguleringen går fra en høyere til laverese tilstand. (tining -> standby, standby -> av)", text variable: PLC_PRG.hysterese_C
        OnMouseClick: write the text variable via VisuDialogs.Numpad
    Textfield (20,299 186x30), "Nedre grense for tining aktiv: %s", text variable: PLC_PRG.min_temp_aktiv
        toggle PLC_PRG.min_temp_aktiv
    Textfield (20,339 186x30), "Nedre grense for tining: %s", text variable: PLC_PRG.min_temp_grense
        OnMouseClick: write the text variable via VisuDialogs.Numpad
    ComboBoxInteger (254,139 150x30), variable: valgt_pid, text list: 'ValgtPIDVerdier'
    Textfield (438,179 200x30), "Min Treveisventilåpning :%.1f%%", tooltip "0% er helt åpen mot returstrømmen, 100% er helt åpen mot smeltesoner", text variable: PLC_PRG.ventil0_min
        OnMouseClick: write the text variable via VisuDialogs.Numpad, min 0, max PLC_PRG.ventil0_maks
    Textfield (438,139 200x30), "Max Treveisventilåpning :%.1f%%", tooltip "0% er helt åpen mot returstrømmen, 100% er helt åpen mot smeltesoner", text variable: PLC_PRG.ventil0_maks
        OnMouseClick: write the text variable via VisuDialogs.Numpad, min PLC_PRG.ventil0_min, max 100
    Textfield (438,299 200x30), "Grenser for smeltesoneventil %i", tooltip "Velg sonen du ønsker å endre ventilverdier", text variable: valgt_ventil
        OnMouseClick: write the text variable via VisuDialogs.Numpad, min 1, max PLC_PRG.antall_soner
    Textfield (24,475 258x30), "Øvre grense for varmeveksler-sikring: %.1f", tooltip "regulering av treveisventilen vil starte når returstrømmen når denne grensen", text variable: PLC_PRG.veksler_temp_grense
        OnMouseClick: write the text variable via VisuDialogs.Numpad
    Label (75,424 157x30), "Sikringer"
    Textfield (24,515 258x30), "Område for varmevekslesikring: %.1f", tooltip "når retur temp når øvre grense - område for sikring vil treveisventilen være 100% åpen for returstrømmen", text variable: PLC_PRG.temp_beskyttelse_omraade
        OnMouseClick: write the text variable via VisuDialogs.Numpad, min 0
    Textfield (390,641 301x30), "Manuell treveisventil: %s", tooltip "skru manuell styring av/på", text variable: PLC_PRG.manuell0
        toggle PLC_PRG.manuell0
    Textfield (389,681 301x30), "Treveisventilåpning: %.1f%%", text variable: PLC_PRG.bestemt0_aapning
        OnMouseClick: write the text variable via VisuDialogs.Numpad
    Textfield (390,561 300x30), "Valgt ventil: %i", text variable: valgt_ventil
        OnMouseClick: write the text variable via VisuDialogs.Numpad
    Textfield (729,521 258x30), "Prognose forvarmingshorisont: %.1f timer", tooltip "Hvor mange timer framover prognosen skal se", text variable: PLC_PRG.forvarme_horisont
    Label (737,430 235x30), "Prognose kontroll"
    Textfield (732,481 255x30), "Prognose aktiv: %s", tooltip "skru prognose av/på", text variable: PLC_PRG.predikt
        toggle PLC_PRG.predikt
END_VISUALIZATION

(* text list ValgtPIDVerdier (id | default)
  0 | Treveisventil
  1 | Pumpe
  2 | Smeltesoneventiler
   |  *)

(* text list Bakkesensor (id | default)
  0 | Etog-56
  1 | test2
   |  *)

(* text list Energiventil (id | default)
  0 | Belimo
  1 | Siemens
   |  *)

(* text list Pumpe (id | default)
  0 | Grundfos UP 25-80
  1 | Test1
   |  *)
